INTERFACE I_Patlite

METHOD bBuzzer : BOOL
VAR_INPUT
	eMachineState		:E_MachineState;
END_VAR
END_METHOD

METHOD bLED :BOOL
VAR_INPUT
	eMachineState		:E_MachineState;
END_VAR
END_METHOD

PROPERTY bSwitchProp : BOOL
GET
END_GET
END_PROPERTY

END_INTERFACE

(* stored: Version 1.1.0.1, ProductVersion 3.1.4024.12
   Itf I_Patlite: Id {14c97931-95fa-40c6-b082-3bd22a2a5f82}
   Method bBuzzer: Id {23f2bed4-27e7-4078-b5ce-6129bab22e71}
   Method bLED: Id {48fbf73f-125a-4d59-b845-3102cbd4b216}
   Property bSwitchProp: Id {9da53c8a-8b53-4b14-8a56-c55a59ce11be}
   Get Get: Id {ca6211ca-c152-4ad4-b15c-1775093ed080} *)
